FUNCTION_BLOCK fb_test
VAR_INPUT
END_VAR
VAR_OUTPUT
END_VAR
VAR
END_VAR

END_FUNCTION_BLOCK

(* stored: Version 1.1.0.1, ProductVersion 3.1.4024.12
   POU fb_test: Id {b52271f6-142e-4284-8dab-062fe243e4d2}, SpecialFunc None *)
